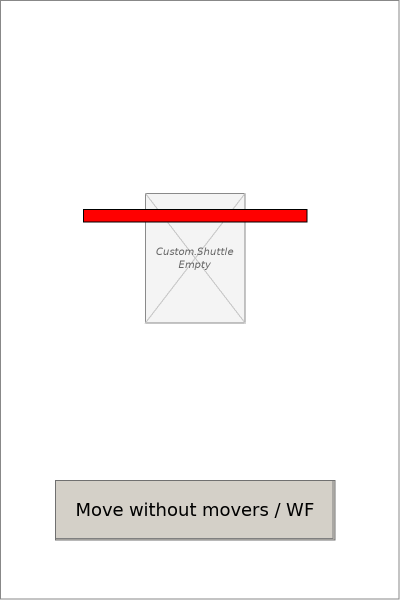
VISUALIZATION VISU_ST128  // 400x600
    Image (145,193 100x130), invisible if: NOT __ISVALIDREF(GVL.st128_aut._Mover), image: Custom.Shuttle Empty
        p2738717112: GVL.st128_aut.fb_TubeCapCheck.visu_shuttle_x_position
    Button (55,480 280x60), "Move without movers / WF", colour toggle: HMI.bArForceCyclusState[StationList_e.ST128]
        tap HMI.btArForceCyclus[StationList_e.ST128].button
    Rectangle (83,209 224x13)
END_VISUALIZATION

(* stored: Version 1.1.0.1, ProductVersion 3.1.4024.6
   Visu VISU_ST128: Id {71c46d88-e52a-4886-a88b-4d491f13dbbb} *)
